FUNCTION_BLOCK PAEElevator EXTENDS PAETransport
VAR_INPUT
END_VAR
VAR_OUTPUT
END_VAR
VAR
END_VAR

END_FUNCTION_BLOCK

(* stored: Version 1.1.0.1, ProductVersion 3.1.4020.12
   POU PAEElevator: Id {6d6b7513-06e2-46f7-a163-9a60ec1ee371}, SpecialFunc None *)
